// TIA Portal V20 export
TYPE "typeIntConditionHmiInterface"
// stored: Access Published, Namespace Unit1.Em5
   STRUCT
      Axis_11 { S7_SetPoint := 'True'} : "LER_typeAxisIntlockAll";   // AnodeMainPnP1AxisX
      Axis_12 { S7_SetPoint := 'True'} : "LER_typeAxisIntlockAll";   // AnodeMainPnP2AxisX
      Axis_13 { S7_SetPoint := 'True'} : "LER_typeAxisIntlockAll";
      Axis_14 { S7_SetPoint := 'True'} : "LER_typeAxisIntlockAll";
      Axis_15 { S7_SetPoint := 'True'} : "LER_typeAxisIntlockAll";
      Axis_16 { S7_SetPoint := 'True'} : "LER_typeAxisIntlockAll";
      Actuator_42 { S7_SetPoint := 'True'} : "LER_typeAxisActuatorCondition";   // AnodeNgBoxLockUpDown
      Actuator_43 { S7_SetPoint := 'True'} : "LER_typeAxisActuatorCondition";   // AnodeMaintenanceMovingFixFrontFwdBwd
   END_STRUCT;
END_TYPE
